TYPE UDPClientOutputStatus_typ :
STRUCT
		opened : BOOL;	
END_STRUCT
END_TYPE

(* stored: Version 1.1.0.1, ProductVersion 3.1.4024.3
   DUT UDPClientOutputStatus_typ: Id {fd54b79a-dadf-0522-17af-84ce11786065} *)
